TEXTLIST MoverMode_TXT
  1 = 'Individual'
  2 = 'Double'
  3 = 'Triple'
   = ''
END_TEXTLIST

(* stored: Version 1.1.0.1, ProductVersion 3.1.4024.11
   TextList MoverMode_TXT: Id {982ab954-d3b1-4244-9af8-19fe3b2c6457} *)
